# EPICS autosave request: iocBoot/sioc-in10-bl01/blen_manual.req
file "manual.req" AREA=IN10,POS=596,INST=BZ10596A
file "manual.req" AREA=IN10,POS=596,INST=BZ10596B
